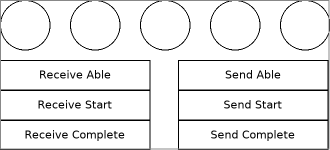
VISUALIZATION Unit  // 330x150
VAR_IN_OUT
	fbUnit : FB_Unit;
END_VAR
    Ellipse (0,0 50x50), invisible if: fbUnit.Inactive
        toggle fbUnit.LED[0]
    Ellipse (70,0 50x50), invisible if: fbUnit.Inactive
        toggle fbUnit.LED[1]
    Ellipse (140,0 50x50), invisible if: fbUnit.Inactive
        toggle fbUnit.LED[2]
    Ellipse (210,0 50x50), invisible if: fbUnit.Inactive
        toggle fbUnit.LED[3]
    Ellipse (280,0 50x50), invisible if: fbUnit.Inactive
        tap fbUnit.LED[4]
    Rectangle (0,60 150x30), "Receive Able", colour toggle: fbUnit._Receivable, invisible if: fbUnit.Inactive
    Rectangle (0,90 150x30), "Receive Start", colour toggle: fbUnit._ReceiveStart, invisible if: fbUnit.Inactive
    Rectangle (0,120 150x30), "Receive Complete", colour toggle: fbUnit._ReceiveComplete, invisible if: fbUnit.Inactive
    Rectangle (178,60 150x30), "Send Able", colour toggle: fbUnit._Sendable, invisible if: fbUnit.Inactive
    Rectangle (178,90 150x30), "Send Start", colour toggle: fbUnit._SendStart, invisible if: fbUnit.Inactive
    Rectangle (178,120 150x30), "Send Complete", colour toggle: fbUnit._SendComplete, invisible if: fbUnit.Inactive
END_VISUALIZATION

(* stored: Version 1.1.0.1, ProductVersion 3.1.4024.12
   Visu Unit: Id {68a63d64-710b-4ca9-beee-208b3a7619f0} *)
